(* IEC 61131-3 sources: plc_on_fpga_riscv_hybrid/RV_FPGA_PLC_IDE_Projects/Basic_IO, 1 file *)

(* ---- Basic_IO.il ---- *)
VAR
END_VAR

PROGRAM Basic_IO
    R1 :
        LD     %SW.0
        ST     %LEDG.0
END_PROGRAM
